(* PLC project static_torsion.project, CODESYS CODESYS V3.5 SP17 Patch 3 *)
(* stored: creationDateTime 1970-01-01T00:00:00, modificationDateTime 2026-06-22T15:12:39.4699931 *)

FUNCTION _dint_to_word2 : ARRAY[0..1] OF WORD
  VAR_INPUT
    _dint : UDINT;
  END_VAR
  VAR
    p_int : POINTER TO UDINT;
    p_words : POINTER TO ARRAY[0..1] OF WORD;
  END_VAR

            p_int := ADR(_dint);
p_words := p_int;
_dint_to_word2 := p_words^;
          
END_FUNCTION
